// Load stacker HW inputs
TYPE ST_HW_InputsMovableStop :
STRUCT	
	LiftUp		: BOOL;		// Sensor inputs 
	LiftDown	: BOOL;		// Sensor inputs 	

END_STRUCT
END_TYPE

(* stored: Version 1.1.0.1, ProductVersion 3.1.4024.9
   DUT ST_HW_InputsMovableStop: Id {067b1e0f-c5fa-49cf-8de6-ea4d25f56204} *)
